// TIA Portal V19 export
FUNCTION "AreaGen_SafetyInterface_Call" : Void   // FC194, LAD
// stored: Access Published, SetENOAutomatically false
BEGIN

REGION Network 1: Call
   // AreaGen_SafetyInterface
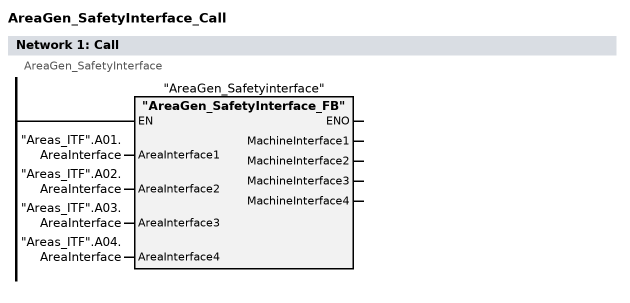
   RUNG wire#powerrail
      "AreaGen_Safetyinterface"(AreaInterface1 := "Areas_ITF".A01.AreaInterface, AreaInterface2 := "Areas_ITF".A02.AreaInterface, AreaInterface3 := "Areas_ITF".A03.AreaInterface, AreaInterface4 := "Areas_ITF".A04.AreaInterface, MachineInterface1 =>, MachineInterface2 =>, MachineInterface3 =>, MachineInterface4 =>)
   END_RUNG
   // the same network as SCL:
   "AreaGen_Safetyinterface"(AreaInterface1 := "Areas_ITF".A01.AreaInterface,   // "AreaGen_SafetyInterface_FB"
                           AreaInterface2 := "Areas_ITF".A02.AreaInterface,
                           AreaInterface3 := "Areas_ITF".A03.AreaInterface,
                           AreaInterface4 := "Areas_ITF".A04.AreaInterface);
END_REGION
END_FUNCTION
